{attribute 'GeneratedUsingTerminal: KL1859'}
{attribute addProperty BoxType "KL1859"}
{attribute addProperty Id "Channel_1AT %Q*Channel_70C997F30Channel_2AT %Q*Channel_70C997F30Channel_3AT %Q*Channel_70C997F30Channel_4AT %Q*Channel_70C997F30Channel_5AT %Q*Channel_70C997F30Channel_6AT %Q*Channel_70C997F30Channel_7AT %Q*Channel_70C997F30Channel_8AT %Q*Channel_70C997F30"}
{attribute addProperty CRC "3316818018"}
{attribute addProperty Size "0"}
TYPE KL1859_C5B2A062 :
STRUCT
	{attribute addProperty Name "Channel_1"}
	Channel_1 : Channel_70C997F3;
	{attribute addProperty Name "Channel_2"}
	Channel_2 : Channel_70C997F3;
	{attribute addProperty Name "Channel_3"}
	Channel_3 : Channel_70C997F3;
	{attribute addProperty Name "Channel_4"}
	Channel_4 : Channel_70C997F3;
	{attribute addProperty Name "Channel_5"}
	Channel_5 : Channel_70C997F3;
	{attribute addProperty Name "Channel_6"}
	Channel_6 : Channel_70C997F3;
	{attribute addProperty Name "Channel_7"}
	Channel_7 : Channel_70C997F3;
	{attribute addProperty Name "Channel_8"}
	Channel_8 : Channel_70C997F3;
END_STRUCT
END_TYPE

(* stored: Version 1.2.0.0, ProductVersion 3.1.4024.9
   DUT KL1859_C5B2A062: Id {2f7cca90-a229-4f6a-83fd-74fce3db899e} *)
